{attribute 'GeneratedUsingTerminal: EP9128-0020-0016'}
{attribute addProperty BoxType "EP9128-0020-0016"}
{attribute addProperty Id "EtcSlaveTerminalBaseInfoDataAT %I*InfoData_6F19DB2B2"}
{attribute addProperty CRC "2874840167"}
{attribute addProperty Size "2"}
TYPE EP9128_AB5A9467 EXTENDS EtcSlaveTerminalBase :
STRUCT
	{attribute addProperty Name "InfoData"}
	InfoData : InfoData_6F19DB2B;
END_STRUCT
END_TYPE

(* stored: Version 1.2.0.0, ProductVersion 3.1.4024.9
   DUT EP9128_AB5A9467: Id {9d137b67-55bd-4a06-a3d4-dc76ec8c3da8} *)
